FUNCTION_BLOCK WKPC_EMIT (* Periodic Workpiece Emitter *)
  (* Standard: 61499-1; Classification: Simulation *)
  (* Version 0.2, 2004-09-16, JHC, Rockwell Automation, Generalized from PR_EMIT. *)
  (* Version 0.1, 2004-08-06, JHC, Rockwell Automation, Changed PPEG to UINT. *)
  (* Version 0.0, 2002-04-11, JHC, Rockwell Automation *)
  (* Compiler header: package fb.rt.mva; *)
  (* Compiler Java Sun JDK 1.4.2 *)
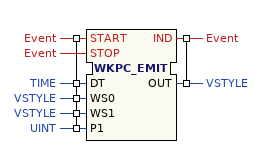
  EVENT_INPUT
    START WITH DT, WS0, WS1, P1; (* Start Periodic Emission *)
    STOP; (* Stop Emission *)
  END_EVENT
  EVENT_OUTPUT
    IND WITH OUT; (* Emission event *)
  END_EVENT
  VAR_INPUT
    DT : TIME := t#6500ms; (* Emission period *)
    WS0 : VSTYLE := PEG; (* Workpiece Style 0 *)
    WS1 : VSTYLE := RING; (* Workpiece Style 1 *)
    P1 : UINT := 50; (* Probability that OUT=WS1 (0-100%) *)
  END_VAR
  VAR_OUTPUT
    OUT : VSTYLE := RING; (* PEG or RING *)
  END_VAR
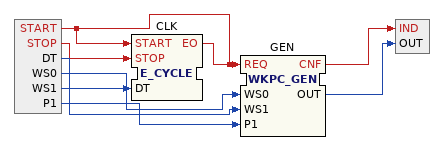
  FBS
    CLK : E_CYCLE;
    GEN : WKPC_GEN;
  END_FBS
  EVENT_CONNECTIONS
    START TO CLK.START;
    STOP TO CLK.STOP;
    CLK.EO TO GEN.REQ;
    START TO GEN.REQ;
    GEN.CNF TO IND;
  END_CONNECTIONS
  DATA_CONNECTIONS
    DT TO CLK.DT;
    GEN.OUT TO OUT;
    WS0 TO GEN.WS0;
    WS1 TO GEN.WS1;
    P1 TO GEN.P1;
  END_CONNECTIONS
END_FUNCTION_BLOCK
